// Mitsubishi GX Works2 project: 双线圈的一些解决办法   PLC: FX3G

// global labels: Global1
VAR_GLOBAL
  真空线圈 AT Y000 : BOOL;
  气缸线圈 AT Y001 : BOOL;
END_VAR

PROGRAM MAIN
VAR
  数据原位_1 : 数据原位;
  真空吸气缸下降_1 : 真空吸气缸下降;
  气缸上升真空破_1 : 气缸上升真空破;
  气缸下降破真空_1 : 气缸下降破真空;
END_VAR
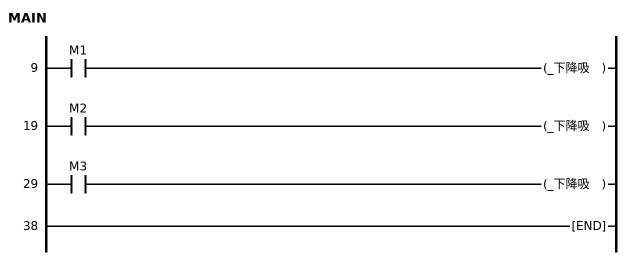
; FB BLK START 数据原位(数据原位_1)
; FB START
; FB_NAME 数据原位
; INSTANCE_NAME 数据原位_1
; FB IN_B:inout
; FB OUT_inout:B
; FB END
; FB BLK END
; FB BLK START 真空吸气缸下降(真空吸气缸下降_1)
9     LD      M1
      OUT     _下降吸
; FB START
; FB_NAME 真空吸气缸下降
; INSTANCE_NAME 真空吸气缸下降_1
; FB IN_B:下降吸
; FB OUT_正常中:B
; FB END
; FB BLK END
; FB BLK START 气缸上升真空破(气缸上升真空破_1)
19    LD      M2
      OUT     _下降吸
; FB START
; FB_NAME 气缸上升真空破
; INSTANCE_NAME 气缸上升真空破_1
; FB IN_B:下降吸
; FB OUT_正常中:B
; FB END
; FB BLK END
; FB BLK START 气缸下降破真空(气缸下降破真空_1)
29    LD      M3
      OUT     _下降吸
; FB START
; FB_NAME 气缸下降破真空
; INSTANCE_NAME 气缸下降破真空_1
; FB IN_B:下降吸
; FB OUT_正常中:B
; FB END
; FB BLK END
38    END
END_PROGRAM

FUNCTION_BLOCK 真空吸气缸下降
VAR_INPUT
  下降吸 : BOOL;
END_VAR
VAR_OUTPUT
  正常中 : BOOL;
END_VAR
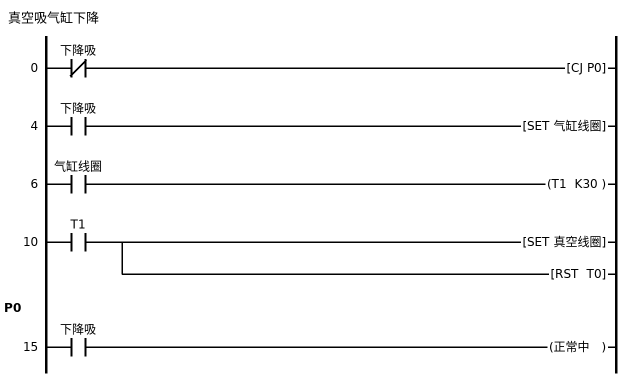
0     LDI     下降吸
      CJ      P0
4     LD      下降吸
      SET     气缸线圈
6     LD      气缸线圈
      OUT     T1 K30
10    LD      T1
      SET     真空线圈
      RST     T0
      P0
15    LD      下降吸
      OUT     正常中
END_FUNCTION_BLOCK

FUNCTION_BLOCK 气缸上升真空破
VAR_OUTPUT
  正常中 : BOOL;
END_VAR
VAR_INPUT
  下降吸 : BOOL;
END_VAR
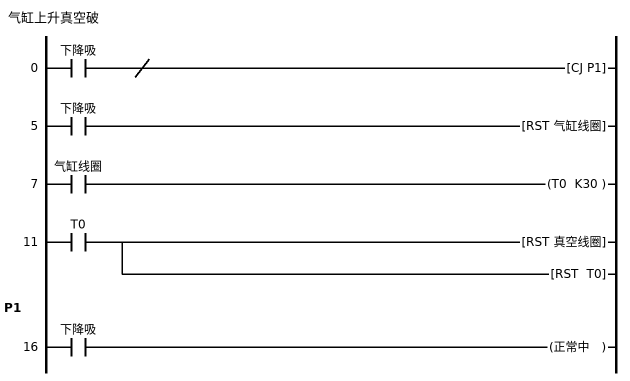
0     LD      下降吸
      INV
      CJ      P1
5     LD      下降吸
      RST     气缸线圈
7     LD      气缸线圈
      OUT     T0 K30
11    LD      T0
      RST     真空线圈
      RST     T0
      P1
16    LD      下降吸
      OUT     正常中
END_FUNCTION_BLOCK

FUNCTION_BLOCK 数据原位
VAR_IN_OUT
  inout : BOOL;
END_VAR
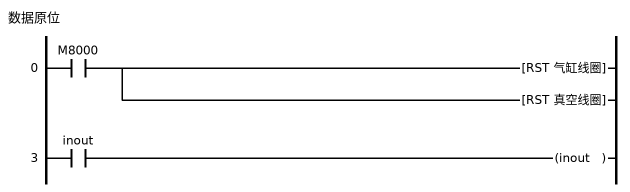
0     LD      M8000
      RST     气缸线圈
      RST     真空线圈
3     LD      inout
      OUT     inout
END_FUNCTION_BLOCK

FUNCTION_BLOCK 气缸下降破真空
VAR_OUTPUT
  正常中 : BOOL;
END_VAR
VAR_INPUT
  下降吸 : BOOL;
END_VAR
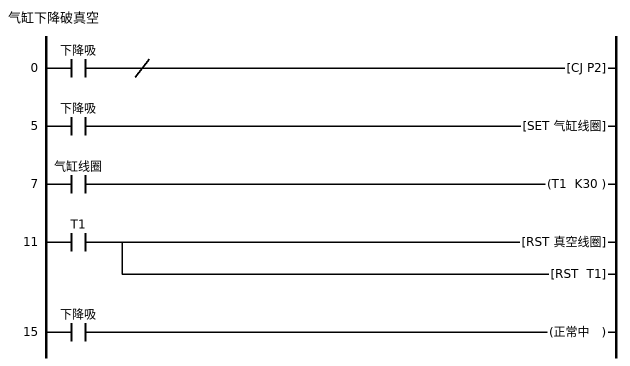
0     LD      下降吸
      INV
      CJ      P2
5     LD      下降吸
      SET     气缸线圈
7     LD      气缸线圈
      OUT     T1 K30
11    LD      T1
      RST     真空线圈
      RST     T1
15    LD      下降吸
      OUT     正常中
      P2
END_FUNCTION_BLOCK
